{attribute 'qualified_only'}
{attribute 'strict'}
TYPE E_CNC_HomingMethod :
(
	Homing		:=  0,
	Measurment	:=  1
)USINT;
END_TYPE

(* stored: Version 1.1.0.1, ProductVersion 3.1.4024.3
   DUT E_CNC_HomingMethod: Id {a88c2396-9209-4ac5-8ee2-daed0be37b68} *)
